INTERFACE I_Message EXTENDS __System.IQueryInterface

// Calculates the size of this message in Protocol Buffer wire format, in bytes.
METHOD CalculateSize : UDINT
VAR_INPUT
END_VAR
END_METHOD

// Merges the data from the specified coded input stream with the current message.
METHOD MergeFrom : HRESULT
VAR_IN_OUT
    fbParseCtx   : FB_ParseContext;
END_VAR
END_METHOD

PROPERTY INTERNAL MessageValue : T_Any
GET
END_GET
END_PROPERTY

/// Parser for this message.
PROPERTY Parser : REFERENCE TO FB_MessageParser
GET
END_GET
END_PROPERTY

/// Writer for this message.
PROPERTY Writer : REFERENCE TO FB_MessageWriter
GET
END_GET
END_PROPERTY

// Writes the data to the given coded output stream.
METHOD WriteTo : HRESULT
VAR_IN_OUT
    fbWriteCtx	: FB_WriteContext;
END_VAR
END_METHOD

END_INTERFACE

(* stored: Version 1.1.0.1
   Itf I_Message: Id {661c5d63-aac8-4fbe-8595-833042ab407b}
   Method CalculateSize: Id {9db2928f-9677-4919-b193-b2e353fc53fc}
   Method MergeFrom: Id {f0218577-d1f3-43ba-b044-8051c53ae231}
   Property MessageValue: Id {97215d09-def5-4507-9b56-dccf22e0973a}
   Get Get: Id {60067ca2-40f7-4972-b244-de71a629b7b8}
   Property Parser: Id {6ab92ca8-0868-416c-9525-df470c1a881e}
   Get Get: Id {9fc93d54-5f70-4bec-980e-8ce0de368e72}
   Property Writer: Id {29b67140-1218-4855-b8d2-0afee340a134}
   Get Get: Id {24e7c725-1dc3-4f60-af6a-1ae67bafdcea}
   Method WriteTo: Id {db7a2abd-e786-44cf-afdc-29280be946e5} *)
